// TIA Portal V18 export
DATA_BLOCK "ST10_Stopper_FB_DB"   // DB1160
// stored: AutoNumber false, InstanceOfName ST10_Stopper_FB, InstanceOfType FB
"ST10_Stopper_FB"
   // VAR
   //    FB_Stopper_Instance { S7_SetPoint := 'True'} : Array[1..3] of "FB_Stopper";
   // END_VAR
BEGIN
END_DATA_BLOCK
